INTERFACE I_CommandFeedback

PROPERTY Aborted : BOOL
GET
END_GET
END_PROPERTY

PROPERTY Busy : BOOL
GET
END_GET
END_PROPERTY

PROPERTY Done : BOOL
GET
END_GET
END_PROPERTY

PROPERTY Error : BOOL
GET
END_GET
END_PROPERTY

PROPERTY PUBLIC ErrorId : UDINT
GET
END_GET
END_PROPERTY

END_INTERFACE

(* stored: Version 1.1.0.1, ProductVersion 3.1.4024.11
   Itf I_CommandFeedback: Id {e5af31a4-1f87-4894-a662-036cfe781cc3}
   Property Aborted: Id {533989e9-7e89-4202-bf14-db277aaad0a4}
   Get Get: Id {dbdfc651-d186-4997-8ba8-51c48b2e9efe}
   Property Busy: Id {3f33c681-b452-4588-8715-8ae3fe0b4969}
   Get Get: Id {5edb1290-036b-4b21-8859-9ee5d40b3ddd}
   Property Done: Id {d3028795-8843-4fd9-b285-59368d0b863b}
   Get Get: Id {bb24b7aa-4482-4f20-b310-4183ac8c2d06}
   Property Error: Id {b3cfd3e9-b669-4bbf-8f47-b0371e7714f2}
   Get Get: Id {f0db0610-b685-417c-8ad3-587376365c11}
   Property ErrorId: Id {7b1acd9c-7db6-4f0a-82f6-f26ace287ef7}
   Get Get: Id {d1d4fbd5-270a-4c52-929b-96fd43dbe6b2} *)
